FUNCTION_BLOCK FB_Conveyor_SFC EXTENDS FB_Object_Template_SFC
VAR_INPUT
	
	END_Conv2:BOOL;

END_VAR
VAR_OUTPUT
	
	MOV_Conv1:BOOL;
	MOV_Conv2:BOOL;

END_VAR
VAR
END_VAR

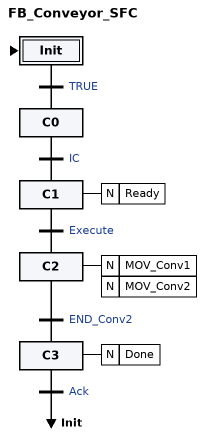
INITIAL_STEP Init:
END_STEP
TRANSITION FROM Init TO C0
    := TRUE;
END_TRANSITION
STEP C0:
END_STEP
TRANSITION FROM C0 TO C1
    := IC;
END_TRANSITION
STEP C1:
    Ready(N);
END_STEP
TRANSITION FROM C1 TO C2
    := Execute;
END_TRANSITION
STEP C2:
    MOV_Conv1(N);
    MOV_Conv2(N);
END_STEP
TRANSITION FROM C2 TO C3
    := END_Conv2;
END_TRANSITION
STEP C3:
    Done(N);
END_STEP
TRANSITION FROM C3 TO Init
    := Ack;
END_TRANSITION

END_FUNCTION_BLOCK

(* stored: Version 1.1.0.1, ProductVersion 3.1.4024.6
   POU FB_Conveyor_SFC: Id {ba4b1948-3804-4c46-bc43-3e685f43d97e}, SpecialFunc None *)
